FUNCTION_BLOCK FB_FireDetection
VAR_IN_OUT CONSTANT
	st_params	: ST_Firedetection_params;
END_VAR

VAR_OUTPUT
	get						:	ST_FireDetection_get;
END_VAR

VAR_OUTPUT	
	b_SystemShutdownCMD 	: 	BOOL;
END_VAR

VAR_INPUT
	Set						:	ST_FireDetection_Set;
	b_BatteryAlarm			: 	BOOL;
END_VAR

VAR	
	b_FireAlarm				: 	BOOL;
	ton_ShutdownDelay		: 	TON := (PT := T#10S);
	ton_SounderOffReset		: 	TON := (PT := T#1S);
	SmokeDetPowerDownTimer 	: 	TP := (PT := TIME#500MS);
END_VAR

VAR
	IO								: FB_FireDetection_IO;
END_VAR

VAR CONSTANT
	w_ID							: WORD := eObject_ID.FireDetection;
END_VAR

IO(st_params:= st_params);

CheckSmokeDetectors(get.SmokeDetectors);
CheckCODetectors(st_params, get.CODetectors);
SounderBeacon();
SetEvents();

get.b_FireAlarm := (get.CODetectors.State = eCOAlarmStatus.Alarm OR get.SmokeDetectors.State = eSmokeDetectAlarmStatus.Alarm);
ton_ShutdownDelay(IN:= b_BatteryAlarm AND get.b_FireAlarm);
IF ton_ShutdownDelay.Q THEN
	b_SystemShutdownCMD := TRUE;
END_IF

//Smoke detector reset
SmokeDetPowerDownTimer(Q => io.SmokeDetectorOFF);
SmokeDetPowerDownTimer.IN := FALSE;

ton_SounderOffReset(IN:= io.SounderOFF);
IF ton_SounderOffReset.Q THEN
	io.SounderOFF := FALSE;
END_IF

METHOD PRIVATE CheckCODetectors : BOOL
VAR_IN_OUT CONSTANT
	st_params : ST_Firedetection_params;
END_VAR

VAR_IN_OUT
	data			: ST_CODetectors;
END_VAR

VAR_INST
	Warning1Timer	:	TON := (PT := TIME#60S);
	Warning2Timer	:	TON := (PT := TIME#60S);
	ErrorTimer		:	TON := (PT := TIME#10S);	
	b_test			:	BOOL; 
END_VAR

VAR
	CoLevelMean			: REAL;
END_VAR
//actual sensor value already filled in in IO code. Only generate status data here.
//alarm status can not be cleared in this method. only via fb_firedetection.reset method.
//alarm status is te highest status, if true, no work to do here.
//if both sensors are working
CoLevelMean := (io.CODetector[1] + io.CODetector[2]) / 2;
data.Value[0] := SEL(CoLevelMean > 5, CoLevelMean, 0);
data.Value[1] := io.CODetector[1];
data.Value[2] := io.CODetector[2];
data.Value[3] := MAX(io.CODetector[1],io.CODetector[2]);

ErrorTimer		(IN := CoLevelMean > st_params.r_COalarmLevel);
Warning1Timer	(IN := CoLevelMean > st_params.r_COwarningLevel_1);
Warning2Timer	(IN := CoLevelMean > st_params.r_COwarningLevel_2);
	
//sr_COalarmState(Set1:=ErrorTimer.Q OR b_test);
//sr_COalarmState.RESET := FALSE;

IF ErrorTimer.Q THEN
	data.State := eCOAlarmStatus.Alarm;
END_IF
	
IF data.State <> eCOAlarmStatus.Alarm THEN
	IF Warning2Timer.Q THEN
		data.State := eCOAlarmStatus.WarningLevel2;
	ELSIF Warning1Timer.Q THEN
		data.State := eCOAlarmStatus.WarningLevel1;
	ELSIF (io.CODetector[1] = -1) OR (io.CODetector[2] = -1) THEN
		data.State := eCOAlarmStatus.Error;
	ELSE
		data.State := eCOAlarmStatus.Normal;
	END_IF
END_IF

data.b_CoValuesOK := NOT (ErrorTimer.Q OR data.State = eCOAlarmStatus.Error);
END_METHOD

METHOD PRIVATE CheckSmokeDetectors

VAR_IN_OUT
	data : ST_Smokedetectors;
END_VAR

VAR_INST
	AlarmResetTimer: TP := (PT := TIME#500MS);
	SmokeAlarmTimer: TON := (PT := TIME#500ms);
	AlarmResetTrigger: F_TRIG;
	SmokeAlarmPowerLost: TON := (PT := TIME#50MS);
END_VAR
//input delay for alarm inputs
SmokeAlarmTimer(IN := (NOT io.SmokeDetector.Signal_OK) AND (NOT AlarmResetTrigger.Q));
SmokeAlarmPowerLost(IN := (NOT  io.SmokeDetector.Power_OK) AND  (NOT AlarmResetTrigger.Q));

IF data.State = eSmokeDetectAlarmStatus.Normal THEN
	IF SmokeAlarmPowerLost.Q THEN	//Alarm power failure means alarm cannot be trusted. So first check power
		data.State := eSmokeDetectAlarmStatus.Error;
	ELSIF SmokeAlarmTimer.Q THEN	//if alarm signals for >500ms --> raise the alarm.
		data.State := eSmokeDetectAlarmStatus.Alarm;	//alarm is only resettable manually via resetDetectors
	END_IF
ELSIF get.SmokeDetectors.State = eSmokeDetectAlarmStatus.Error THEN	//if power failed, no alarm checking anymore as this will give false alarms
	IF NOT SmokeAlarmPowerLost.Q THEN	//Alarm state may return to operational if power comes back
		data.State := eSmokeDetectAlarmStatus.Normal;
	END_IF
END_IF	//In alarm state, no power checking is performed anymore. Even if the detectors lose power now, the alarm state has priority.
END_METHOD

METHOD PUBLIC EMstop : BOOL
VAR_INPUT
END_VAR
//do anything?
//return true when ready
END_METHOD

METHOD GetDiagnostics
VAR_IN_OUT
	AddError		: ARRAY [*] OF FB_AddErrorST;
	a_ActiveEvents	: ARRAY [*] OF ST_ErrorStruct;
	w_Index			: WORD;
END_VAR
(*Alarm Muted *)		AddError[w_Index](
		b_ErrorTrig			:= get.events.AlarmMuted,
		out_ST_Error			:= a_ActiveEvents[w_Index],
		w_ErrorID					:= 1,
		e_ObjectID				:= eObject_ID.Firedetection,
		s_Message				:= 'alarm muted',
		e_sev					:= eseverity.info,
		b_AutoClear				:= TRUE,
		e_ErrAckAccess		:= eErrAckAccess.General
	);
	w_Index := w_Index +1;

(*Smoke NOK*)			AddError[w_Index](
		b_ErrorTrig			:= get.events.SmokeDetFault,
		out_ST_Error			:= a_ActiveEvents[w_Index],
		w_ErrorID					:= 2,
		s_Message				:= 'smoke detector not OK',
		e_sev					:= eseverity.warning,
		t_triggerTime			:= T#5S,
		b_AutoClear				:= TRUE,
		e_ErrAckAccess		:= eErrAckAccess.operator,
	);
	w_Index := w_Index +1;

(*Smoke alarm*)			AddError[w_Index](
		b_ErrorTrig				:= get.events.SmokeDetAlarm,
		out_ST_Error			:= a_ActiveEvents[w_Index],
		w_ErrorID				:= 3,
		s_Message				:= 'smoke detector alarm',
		e_sev					:= eseverity.Quickshutdown,
		e_ErrAckAccess			:= eErrAckAccess.VDL,
		b_SMSEnableVDL			:= TRUE,
	);
	w_Index := w_Index +1;

(*CO NOK*)				AddError[w_Index](
		b_ErrorTrig				:= get.events.CODetFault,
		out_ST_Error			:= a_ActiveEvents[w_Index],
		w_ErrorID				:= 4,
		s_Message				:= 'CO detector not OK',
		e_sev					:= eseverity.Warning,
		b_AutoClear				:= TRUE,
		e_ErrAckAccess			:= eErrAckAccess.operator,
		t_TriggerTime			:= T#2S,
	);
	w_Index := w_Index +1;

(*CO warning level1*)			AddError[w_Index](
		b_ErrorTrig				:= get.events.CODetWarning1,
		out_ST_Error			:= a_ActiveEvents[w_Index],
		w_ErrorID				:= 5,
		s_Message				:= CONCAT(CONCAT('CO Detector warning level 1: ', TO_STRING(st_params.r_COwarningLevel_1)), ' ppm'),
		e_sev					:= eseverity.info,
		e_ErrAckAccess			:= eErrAckAccess.Operator,
		b_AutoClear				:= TRUE,
		b_SMSEnableVDL			:= FALSE,
	);
	w_Index := w_Index +1;
	
(*CO warning level2*)			AddError[w_Index](
		b_ErrorTrig				:= get.events.CODetWarning2,
		out_ST_Error			:= a_ActiveEvents[w_Index],
		w_ErrorID				:= 6,
		s_Message				:= CONCAT(CONCAT('CO Detector warning level 2: ', TO_STRING(st_params.r_COwarningLevel_2)), ' ppm'),
		e_sev					:= eseverity.Warning,
		e_ErrAckAccess			:= eErrAckAccess.operator,
		b_AutoClear				:= TRUE,
		b_SMSEnableVDL			:= FALSE,
	);
	w_Index := w_Index +1;

(*CO alarm*)			AddError[w_Index](
		b_ErrorTrig				:= get.events.CODetAlarm,
		out_ST_Error			:= a_ActiveEvents[w_Index],
		w_ErrorID				:= 7,
		s_Message				:=  CONCAT(CONCAT('CO Detector alarm level: ', TO_STRING(st_params.r_COAlarmLevel)), ' ppm'),
		e_sev					:= eseverity.NormalShutdown,
		e_ErrAckAccess			:= eErrAckAccess.VDL,
		b_SMSEnableVDL			:= TRUE,
	);
	w_Index := w_Index +1;
END_METHOD

METHOD PUBLIC Reset : BOOL
VAR_INPUT
//	ResetActive : BOOL := FALSE;
END_VAR

VAR_INST
	b_status : BOOL;
END_VAR
//return true when ready



IF io.smokedetector.Power_OK AND io.smokedetector.Signal_OK THEN
	get.SmokeDetectors.State := eSmokeDetectAlarmStatus.Normal;
END_IF

IF get.CODetectors.b_CoValuesOK THEN
	get.CODetectors.State := eCOAlarmStatus.Normal;
END_IF

b_status := get.CODetectors.State = eCOAlarmStatus.Normal AND get.SmokeDetectors.State = eSmokeDetectAlarmStatus.Normal;
SmokeDetPowerDownTimer.IN := NOT b_status;

IF b_status THEN
	io.SounderON := FALSE;
	io.SounderOFF := TRUE;
END_IF

Reset := b_status AND io.smokedetector.Power_OK;
END_METHOD

METHOD SetEvents : BOOL
VAR_INPUT
END_VAR
get.Events.SmokeDetAlarm 	:= (get.SmokeDetectors.State = eSmokeDetectAlarmStatus.Alarm);
get.Events.SmokeDetFault 	:= (get.SmokeDetectors.State = eSmokeDetectAlarmStatus.Error);
get.Events.CODetAlarm 		:= (get.CODetectors.State = eCOAlarmStatus.Alarm);
get.Events.CODetFault 		:= (get.CODetectors.State = eCOAlarmStatus.Error);
get.Events.CODetWarning1	:= get.CODetectors.State = eCOAlarmStatus.WarningLevel1;
get.Events.CODetWarning2	:= get.CODetectors.State = eCOAlarmStatus.WarningLevel2;

get.Events.AlarmMuted 		:= (get.Events.SmokeDetAlarm OR get.Events.CODetAlarm) And not io.SounderOn;
END_METHOD

METHOD SounderBeacon : BOOL

VAR_INST
	
	TestTrigger 		: 	R_Trig;
	SmokeAlarmTrigger	:	R_Trig;
	COAlarmTrigger		:	R_trig;
END_VAR

//Only enable sounder at the start of the alarm. Use old_state to determine this.
//This allows for alarm muting and retriggering. 
COAlarmTrigger(clk:=get.CODetectors.State = eCOAlarmStatus.Alarm);
SmokeAlarmTrigger(Clk:= get.SmokeDetectors.State = eSmokeDetectAlarmStatus.Alarm);

//use rtrig to prevent permanent sounding. resilence with muting.
TestTrigger(clk:= set.TestSounder);

//use rtrig to prevent permanent muting.
IF set.SilenceSounder THEN
	io.SounderOn:= FALSE;
	io.SounderOFF := TRUE;
END_IF

IF COAlarmTrigger.q OR SmokeAlarmTrigger.Q OR TestTrigger.Q THEN;
	io.SounderOn:= TRUE;
END_IF
END_METHOD

END_FUNCTION_BLOCK

(* stored: Version 1.1.0.1, ProductVersion 3.1.4026.18
   POU FB_FireDetection: Id {b98e996a-b696-4831-bfb9-9caf729fd2d4}, SpecialFunc None
   Method CheckCODetectors: Id {0d61aa76-96b6-45e8-a408-310074a41bbe}
   Method CheckSmokeDetectors: Id {32b84b62-fec9-4ace-a986-823787861248}
   Method EMstop: Id {d5edf8eb-e666-4e22-a7b2-96f4ec1cbbc7}
   Method GetDiagnostics: Id {3ac1670d-7016-45f8-8db1-77c0c1fba044}
   Method Reset: Id {4f4218f7-8d22-4aef-88b1-0859d0e6c514}
   Method SetEvents: Id {e3b0d513-3355-450a-b970-462e61e901f3}
   Method SounderBeacon: Id {a2411ec0-a4cc-4891-bf7d-27051458cbfd} *)
